FUNCTION_BLOCK deleteme
VAR_INPUT
END_VAR
VAR_OUTPUT
END_VAR
VAR
END_VAR

END_FUNCTION_BLOCK

(* stored: Version 1.1.0.1, ProductVersion 3.1.4024.12
   POU deleteme: Id {07419c8f-447f-4df7-834d-203d44a00868}, SpecialFunc None *)
